FUNCTION_BLOCK FB_HE_SolidAttenuatorHolderMock EXTENDS FB_FalliblePublicMock IMPLEMENTS I_HE_SolidAttenuatorHolder
VAR
    nNumberOfSlots : INT;
    stSettings : ST_HE_SolidAttenuatorHolderSettings;

END_VAR

{warning 'Add method implementation '}
METHOD GetNumberOfSlots : INT
END_METHOD

{warning 'Add method implementation '}
METHOD GetSettings
VAR_IN_OUT
    Settings	: ST_HE_SolidAttenuatorHolderSettings;
END_VAR
END_METHOD

{warning 'Add method implementation '}
METHOD GetSlotAt
VAR_INPUT
    Position	: I_QuantityLREALPublic;
END_VAR
END_METHOD

END_FUNCTION_BLOCK

(* stored: Version 1.1.0.1
   POU FB_HE_SolidAttenuatorHolderMock: Id {97032738-f9d4-4a7b-b0ed-ed2164124302}, SpecialFunc None
   Method GetNumberOfSlots: Id {15e4c3d3-2c46-4d34-b72d-3b65b88630ee}
   Method GetSettings: Id {901c2515-f91d-4b82-8d34-c135b3a11596}
   Method GetSlotAt: Id {18ebd8ca-3da7-40e1-a134-e5fdcbe6ab82} *)
